ABB RobotStudio station: Workshop_RI.rspag

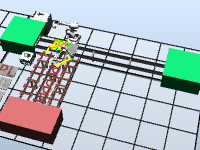
--- station ---
Station Workshop_RI (saved by RobotStudio format 3)
Controller IRB_1600_6kg_1.2m, task T_ROB1: task frame (RAPID world) sits at (2400, 1050, 0) mm, rotated rx 0 ry 0 rz -90 deg in the station
Controller IRB_140_6kg_0.81m, task T_ROB1: task frame (RAPID world) sits at (2400, -400, 420) mm in the station
Controller IRB_140_6kg_0.81m
  mechanical unit ROB_1: IRB140_6_81_C_03, 6 joints, base frame (0, 0, 0) mm
Controller IRB_1600_6kg_1.2m
  mechanical unit ROB_1: IRB1600_6_120__02, 6 joints, base frame (0, 0, 0) mm
Layout (positions relative to the parent item):
  - SC_SimpleVacuumGripper [protected smart component, left out]
  - Backup_Base_Parts [graphiccomponentgroup] at (1500, 500, 0) mm, rotated rx 0 ry 0 rz -90 deg
    - I_color [part] at (1567.69, 3594.7, 0) mm, rotated rx 0 ry 0 rz 90 deg
    - P_color [part] at (1567.69, 3594.7, 0) mm, rotated rx 0 ry 0 rz 90 deg
    - I_org [part] at (2207.69, 3594.7, 0) mm, rotated rx 0 ry 0 rz 90 deg
    - P_org [part] at (2207.69, 3594.7, 0) mm, rotated rx 0 ry 0 rz 90 deg
    - L_org [part] at (2207.69, 3594.7, 0) mm, rotated rx 0 ry 0 rz 90 deg
    - Base_org [part] at (2087.69, -1721.31, 0) mm
    - Base_holes [part] at (1447.69, -1721.31, 0) mm
    - L_color [part] at (1567.69, 3594.7, 0) mm, rotated rx 0 ry 0 rz 90 deg
  - SC_Main_Conveyor [protected smart component, left out]
  - Middle_PlaneSensor [smart component, from Libraries\PlaneSensor.rslib]
      properties: Origin=[2.865 -0.086804 0.458]; Axis1=[0 0.64 0]; Axis2=[0 0 0.05]; SensedPart=Base_holes_42
    - _sensorPart_ [part]
  - TempParts [graphiccomponentgroup]
    - Base_holes_42 [part] at (2866.18, 496.99, 457) mm, rotated rx 0 ry 0 rz 180 deg
    - Base_holes_1 [part] at (180, -43.01, 457) mm
  - SC_Letter_Conveyor_I [protected smart component, left out]
  - AW_Gun_PSF_25 [mechanism, from Tools\AW_Gun_PSF_25.rslib] at (1846.39, 1050, 893.77) mm, rotated rx -180 ry 60 rz 0 deg
  - Teste_Group1 [graphiccomponentgroup]
    - I_color_3 [part] at (7151.02, 376.99, 457) mm
    - L_color [part] at (7151.02, 376.99, 457) mm
    - P_color [part] at (7151.02, 376.99, 457) mm
    - Base_org_332 [part] at (2865, -43.01, 457) mm, rotated rx 0 ry 0 rz 90 deg
  - Teste_Group2 [graphiccomponentgroup] at (1650, 0, 0) mm
    - I_color_3 [part] at (7151.02, 376.99, 457) mm
    - L_color [part] at (7151.02, 376.99, 457) mm
    - P_color [part] at (7151.02, 376.99, 457) mm
    - Base_org_332 [part] at (2865, -43.01, 457) mm, rotated rx 0 ry 0 rz 90 deg
  - Furniture [graphiccomponentgroup]
    - Box_2 [part]
    - Box_3 [part]
    - Table [part] at (1825, -4950, 0) mm, rotated rx 0 ry 0 rz 90 deg
    - FlexPendant [part, from Equipment\FlexPendant.rslib] at (848.68, 1513.9, 739.04) mm, rotated rx -28.56 ry 0 rz 180 deg
    - IRC5_Compact [part, from Equipment\IRC5_Compact__02.rslib] at (772.3, -736.92, 0) mm
    - IRC5_Control-Module [part, from Equipment\IRC5_Control-Module.rslib] at (873.2, 1576.94, 100) mm, rotated rx 90 ry 0 rz 180 deg
    - FlexPendant_2 [part, from Equipment\FlexPendant.rslib] at (1028.44, -563.39, 415.73) mm, rotated rx -28.56 ry 0 rz 0 deg
  - IRB140_6_81_C_03 [mechanism, from Robots\IRB140_6_81_C_G_03.rslib] at (2400, -400, 420) mm; joint values [0, 0.4698, 0.3639, 0, 0.5236, 0] (rad or m)
  - SC_Letter_Conveyor_P [protected smart component, left out]
  - SC_Letter_Conveyor_L [protected smart component, left out]
  - Part_12 [part]
  - IRB1600_6_120__02 [mechanism, from Robots\IRB1600_6_120_G_02.rslib] at (2400, 1050, 0) mm, rotated rx 0 ry 0 rz -90 deg; joint values [-1.5708, -0.5581, 0.4967, 0, 0.5851, 0] (rad or m)
Attachment: SC_SimpleVacuumGripper is attached to IRB140_6_81_C_03 / Link6
Attachment: AW_Gun_PSF_25 is attached to IRB1600_6_120__02 / Link6
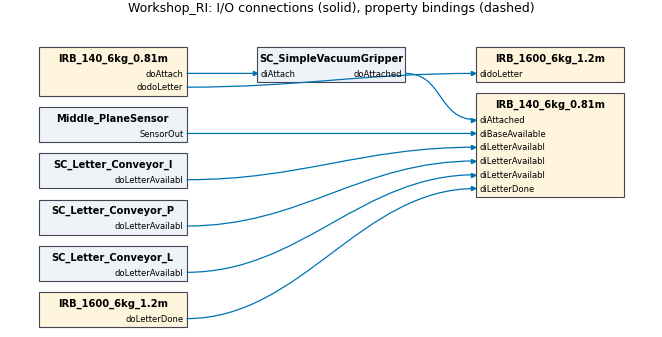
Station logic (signal -> signal, property => property):
  IRB_140_6kg_0.81m.doAttach -> SC_SimpleVacuumGripper.diAttach
  SC_SimpleVacuumGripper.doAttached -> IRB_140_6kg_0.81m.diAttached
  Middle_PlaneSensor.SensorOut -> IRB_140_6kg_0.81m.diBaseAvailable
  SC_Letter_Conveyor_I.doLetterAvailable -> IRB_140_6kg_0.81m.diLetterAvailable_I
  SC_Letter_Conveyor_P.doLetterAvailable -> IRB_140_6kg_0.81m.diLetterAvailable_P
  SC_Letter_Conveyor_L.doLetterAvailable -> IRB_140_6kg_0.81m.diLetterAvailable_L
  IRB_140_6kg_0.81m.dodoLetter -> IRB_1600_6kg_1.2m.didoLetter
  IRB_1600_6kg_1.2m.doLetterDone -> IRB_140_6kg_0.81m.diLetterDone

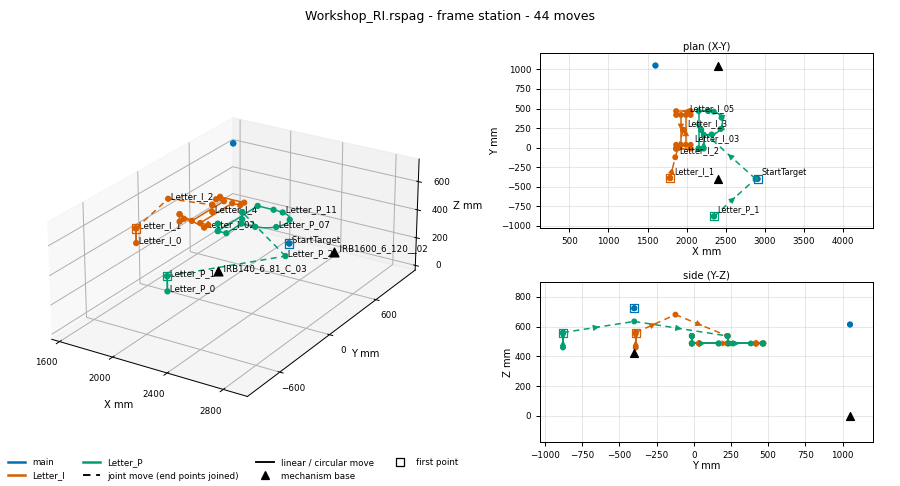
[picture p0: tool path of Workshop_RI.rspag in frame station, 44 of 44 moves have a stored position in this frame; points joined in program order, loops and branches not executed]
--- Backups/IRB_140_6kg_0.81m/RAPID/TASK1/PROGMOD/CalibData.mod ---
MODULE CalibData
	PERS tooldata SimpleVacuumGripper:=[TRUE,[[0,0,25],[1,0,0,0]],[0.5,[0,0,1],[1,0,0,0],0,0,0]];
ENDMODULE

--- Backups/IRB_140_6kg_0.81m/RAPID/TASK1/PROGMOD/Module1.mod ---
MODULE Module1
	CONST robtarget Letter_I_1:=[[-611.4,9.874,140],[0,-0.707106781,0.707106781,0],[1,0,0,0],[9E9,9E9,9E9,9E9,9E9,9E9]];
	CONST robtarget Letter_I_0:=[[-611.4,9.874,40],[0,-0.707106781,0.707106781,0],[1,0,0,0],[9E9,9E9,9E9,9E9,9E9,9E9]];
	CONST robtarget Letter_I_2:=[[-545.231385656,276.821478528,260.515371052],[-0.000000405,-0.529975894,0.848012707,-0.000000052],[1,0,0,0],[9E9,9E9,9E9,9E9,9E9,9E9]];
	CONST robtarget Letter_I_3:=[[-441.034,626.99,117],[0,1,0,0],[1,0,-1,0],[9E9,9E9,9E9,9E9,9E9,9E9]];
	CONST robtarget Letter_I_4:=[[-441.034,626.99,67],[0,1,0,0],[1,0,-1,0],[9E9,9E9,9E9,9E9,9E9,9E9]];
	CONST robtarget Letter_P_1:=[[-50,-479.055,140],[0,-0.707106781,0.707106781,0],[-2,0,1,0],[9E9,9E9,9E9,9E9,9E9,9E9]];
	CONST robtarget Letter_P_0:=[[-50,-479.055,40],[0,-0.707106781,0.707106781,0],[-2,0,1,0],[9E9,9E9,9E9,9E9,9E9,9E9]];
	CONST robtarget Letter_P_2:=[[481.657122129,0,215.039783495],[0.00000001,0.998648416,0.051974428,0.000000187],[0,-1,1,0],[9E9,9E9,9E9,9E9,9E9,9E9]];
	CONST robtarget Letter_P_3:=[[-213.633,626.99,117],[0,1,0,0],[1,0,3,0],[9E9,9E9,9E9,9E9,9E9,9E9]];
	CONST robtarget Letter_P_4:=[[-213.633,626.99,67],[0,1,0,0],[1,0,3,0],[9E9,9E9,9E9,9E9,9E9,9E9]];
    CONST robtarget StartPose:=[[507.45080207,0,303.659048752],[0.106520171,0,0.994310542,0],[0,0,0,0],[9E9,9E9,9E9,9E9,9E9,9E9]];
	CONST robtarget StartTarget:=[[507.45080207,0,303.659048752],[0.106520171,0,0.994310542,0],[0,0,0,0],[9E9,9E9,9E9,9E9,9E9,9E9]];
	PROC main()
        MoveJ StartTarget,v1000,z100,SimpleVacuumGripper\WObj:=wobj0;
        SetDO dodoLetter,0;
        WaitDI diLetterDone,0;
        Letter_I;
		Letter_P;
		Letter_L;
		MoveJ StartTarget,v1000,z100,SimpleVacuumGripper\WObj:=wobj0;
        SetDO dodoLetter,1;
        WaitDI diLetterDone,1;
    ENDPROC
    PROC Letter_I()
	    MoveJ Letter_I_1,v1000,z5,SimpleVacuumGripper\WObj:=wobj0;
	    MoveL Letter_I_0,v100,fine,SimpleVacuumGripper\WObj:=wobj0;
	    SetDO doAttach,1;
	    WaitDI diAttached,1;
	    MoveL Letter_I_1,v100,z10,SimpleVacuumGripper\WObj:=wobj0;
	    MoveJ Letter_I_2,v1000,z100,SimpleVacuumGripper\WObj:=wobj0;
	    MoveJ Letter_I_3,v1000,z5,SimpleVacuumGripper\WObj:=wobj0;
	    MoveL Letter_I_4,v100,fine,SimpleVacuumGripper\WObj:=wobj0;
	    SetDO doAttach,0;
	    WaitDI diAttached,0;
		MoveL Letter_I_3,v100,z5,SimpleVacuumGripper\WObj:=wobj0;
	ENDPROC
	PROC Letter_P()
	    MoveJ Letter_P_1,v1000,z5,SimpleVacuumGripper\WObj:=wobj0;
	    MoveL Letter_P_0,v100,fine,SimpleVacuumGripper\WObj:=wobj0;
	    SetDO doAttach,1;
	    WaitDI diAttached,1;
	    MoveL Letter_P_1,v100,z10,SimpleVacuumGripper\WObj:=wobj0;
	    MoveJ Letter_P_2,v1000,z10,SimpleVacuumGripper\WObj:=wobj0;
	    MoveJ Letter_P_3,v1000,z5,SimpleVacuumGripper\WObj:=wobj0;
	    MoveL Letter_P_4,v100,fine,SimpleVacuumGripper\WObj:=wobj0;
	    SetDO doAttach,0;
	    WaitDI diAttached,0;
		MoveL Letter_P_3,v100,z10,SimpleVacuumGripper\WObj:=wobj0;
	ENDPROC
	PROC Letter_L()
	ENDPROC
ENDMODULE

--- Backups/IRB_140_6kg_0.81m/RAPID/TASK1/SYSMOD/LINKEDM.sys ---
%%%
  VERSION:1
  LANGUAGE:ENGLISH
%%%

MODULE LINKEDM (SYSMODULE)

! FOLLOWER
!     Name of electronically linked follower axis used by operator at teach pendent.
      PERS string l_f_axis_name{5}       :=  ["",  "", "", "", ""];

!     Name of the mechanical unit for follower axis.
      PERS string l_f_mecunt_n{5}  :=  ["", "", "", "", ""];

!     Linked follower axis number in the mechanical unit (first axis in mech. unit is number 1).
      PERS num l_f_axis_no{5}      :=  [0,          0,   0,  0,  0];

! MASTER
!     Name of the mechanical unit for linked master axis.
      PERS string l_m_mecunt_n{5} :=  ["", "", "", "", ""];

!     Linked master axis number in the mechanical unit (first axis in mech. unit is number 1).
!     See axis number table in documentation for different master mechanical units.
      PERS num l_m_axis_no{5}     :=  [0,  0,  0,  0,  0];

! POSITION OFFSET
!     The increase of the allowed offset position between the master and follower
!     positions, used when starting AUTO mode. As soon as the offset is decreased
!     the old configurated parameter is used.
!     Example: 3 => the configurated value of allowed offset is increased 3 times.
      PERS num offset_ratio{5}       :=  [10,  10,   10,  10,  10];

! SPEED RATIO
!     Speed_ratio used in AUTO and JOG modes [ very_slow   slow    normal    fast]
!     Value 1 = max allowed manual speed.
      CONST num speed_ratio {20}      := [0.01, 0.01, 0.01, 0.01, 0.01,
                                          0.05, 0.05, 0.05, 0.05, 0.05,
                                          0.20, 0.20, 0.20, 0.20, 0.20,
                                          1.00, 1.00, 1.00, 1.00, 1.00];

! STEP SIZE
!     Displacement position used in JOG mode for each activation of positive or
!     negative movement.                  [very_short    short   normal   long]
!     Unit degees or meter.
      CONST num displacement {20}     := [0.001, 0.001, 0.001, 0.001, 0.001,
                                          0.005, 0.005, 0.005, 0.005, 0.005,
                                          0.020, 0.020, 0.020, 0.020, 0.020,
                                          0.100, 0.100, 0.100, 0.100, 0.100];


!-------------------------------------------------------------
 PROC Linked_m ()
      Linked_m_exe ;
 ENDPROC
ENDMODULE

--- Backups/IRB_1600_6kg_1.2m/RAPID/TASK1/PROGMOD/CalibData.mod ---
MODULE CalibData
	PERS tooldata AW_Gun:=[TRUE,[[119.5,0,352],[0.890213743,0,0.455543074,0]],[1,[0,0,100],[1,0,0,0],0,0,0]];
ENDMODULE

--- Backups/IRB_1600_6kg_1.2m/RAPID/TASK1/PROGMOD/Module1.mod ---
MODULE Module1
	CONST robtarget Letter_I_00:=[[1063.009551758,-533.999941406,537],[0,0,1,0],[-1,0,-1,0],[9E9,9E9,9E9,9E9,9E9,9E9]];
	CONST robtarget Letter_I_02:=[[1063.009551758,-348.068012719,487],[0,0,1,0],[-1,0,-1,0],[9E9,9E9,9E9,9E9,9E9,9E9]];
	CONST robtarget Letter_I_03:=[[1013.998206539,-348.068012719,487],[0,0,1,0],[-1,0,-1,0],[9E9,9E9,9E9,9E9,9E9,9E9]];
	CONST robtarget Letter_I_04:=[[1013.998206539,-409.137704777,487],[0,0,1,0],[-1,0,-1,0],[9E9,9E9,9E9,9E9,9E9,9E9]];
	CONST robtarget Letter_I_05:=[[632.020896977,-409.137704777,487],[0,0,1,0],[-1,0,-1,0],[9E9,9E9,9E9,9E9,9E9,9E9]];
	CONST robtarget Letter_I_06:=[[632.020896977,-348.068012719,487],[0,0,1,0],[-1,0,-1,0],[9E9,9E9,9E9,9E9,9E9,9E9]];
	CONST robtarget Letter_I_07:=[[583.009551758,-348.068012719,487],[0,0,1,0],[-1,0,-1,0],[9E9,9E9,9E9,9E9,9E9,9E9]];
	CONST robtarget Letter_I_08:=[[583.009551758,-533.999941406,487],[0,0,1,0],[-1,0,-1,0],[9E9,9E9,9E9,9E9,9E9,9E9]];
	CONST robtarget Letter_I_09:=[[632.020896977,-533.999941406,487],[0,0,1,0],[-1,0,-1,0],[9E9,9E9,9E9,9E9,9E9,9E9]];
	CONST robtarget Letter_I_10:=[[632.020896977,-472.930249348,487],[0,0,1,0],[-1,0,-1,0],[9E9,9E9,9E9,9E9,9E9,9E9]];
	CONST robtarget Letter_I_11:=[[1013.998206539,-472.930249348,487],[0,0,1,0],[-1,0,-1,0],[9E9,9E9,9E9,9E9,9E9,9E9]];
	CONST robtarget Letter_I_12:=[[1013.998206539,-533.999941406,487],[0,0,1,0],[-1,0,-1,0],[9E9,9E9,9E9,9E9,9E9,9E9]];
	CONST robtarget Letter_I_01:=[[1063.009551758,-533.999941406,487],[0,0,1,0],[-1,0,-1,0],[9E9,9E9,9E9,9E9,9E9,9E9]];
	CONST robtarget Letter_P_00:=[[1063.009551758,-245.528012719,537],[0,0,1,0],[-1,0,-1,0],[9E9,9E9,9E9,9E9,9E9,9E9]];
	CONST robtarget Letter_P_01:=[[1063.009551758,-245.528012719,487],[0,0,1,0],[-1,0,-1,0],[9E9,9E9,9E9,9E9,9E9,9E9]];
	CONST robtarget Letter_P_02:=[[1063.009551758,-181.735468149,487],[0,0,1,0],[-1,0,-1,0],[9E9,9E9,9E9,9E9,9E9,9E9]];
	CONST robtarget Letter_P_03:=[[884.079243816,-181.735468149,487],[0,0,1,0],[-1,0,-1,0],[9E9,9E9,9E9,9E9,9E9,9E9]];
	CONST robtarget Letter_P_04:=[[884.079243816,-127.667396836,487],[0,0,1,0],[-1,0,-1,0],[9E9,9E9,9E9,9E9,9E9,9E9]];
	CONST robtarget Letter_P_05:=[[880.918790007,-80.746813367,487],[0,0,1,0],[-1,0,-1,0],[9E9,9E9,9E9,9E9,9E9,9E9]];
	CONST robtarget Letter_P_06:=[[855.829649003,-11.216829575,487],[0,0,1,0],[-1,0,-1,0],[9E9,9E9,9E9,9E9,9E9,9E9]];
	CONST robtarget Letter_P_07:=[[812.701610105,33.515747411,487],[0,0,1,0],[0,-1,0,0],[9E9,9E9,9E9,9E9,9E9,9E9]];
	CONST robtarget Letter_P_08:=[[743.07438158,57.182684202,487],[0,0,1,0],[0,-1,0,0],[9E9,9E9,9E9,9E9,9E9,9E9]];
	CONST robtarget Letter_P_09:=[[666.679527447,46.260885174,487],[0,0,1,0],[0,-1,0,0],[9E9,9E9,9E9,9E9,9E9,9E9]];
	CONST robtarget Letter_P_10:=[[612.960929392,0.695650166,487],[0,0,1,0],[0,-1,0,0],[9E9,9E9,9E9,9E9,9E9,9E9]];
	CONST robtarget Letter_P_11:=[[590.011172503,-52.205484356,487],[0,0,1,0],[-1,0,-1,0],[9E9,9E9,9E9,9E9,9E9,9E9]];
	CONST robtarget Letter_P_12:=[[584.759956944,-85.365938165,487],[0,0,1,0],[-1,0,-1,0],[9E9,9E9,9E9,9E9,9E9,9E9]];
	CONST robtarget Letter_P_13:=[[583.009551758,-124.944544324,487],[0,0,1,0],[-1,0,-1,0],[9E9,9E9,9E9,9E9,9E9,9E9]];
	CONST robtarget Letter_P_14:=[[583.009551758,-245.528012719,487],[0,0,1,0],[-1,0,-1,0],[9E9,9E9,9E9,9E9,9E9,9E9]];
	CONST robtarget StartTarget:=[[0.000250725,-798.69947369,614.279917089],[0.035775265,0.706201086,0.706201308,-0.035775276],[-1,-1,-1,0],[9E9,9E9,9E9,9E9,9E9,9E9]];
	PROC main()
        MoveJ StartTarget,v1000,z100,AW_Gun\WObj:=wobj0;
        SetDO doLetterDone,0;
        WaitDI didoLetter,0;
        WaitDI didoLetter,1;
        Letter_I;
        Letter_P;
        Letter_L;
        MoveJ StartTarget,v1000,z100,AW_Gun\WObj:=wobj0;
        SetDO doLetterDone,0;

    ENDPROC
    PROC Letter_I()
	    MoveJ Letter_I_00,v1000,z5,AW_Gun\WObj:=wobj0;
	    MoveL Letter_I_02,v200,z0,AW_Gun\WObj:=wobj0;
	    MoveL Letter_I_03,v200,z0,AW_Gun\WObj:=wobj0;
	    MoveL Letter_I_04,v200,z0,AW_Gun\WObj:=wobj0;
	    MoveL Letter_I_05,v200,z0,AW_Gun\WObj:=wobj0;
	    MoveL Letter_I_06,v200,z0,AW_Gun\WObj:=wobj0;
	    MoveL Letter_I_07,v200,z0,AW_Gun\WObj:=wobj0;
	    MoveL Letter_I_08,v200,z0,AW_Gun\WObj:=wobj0;
	    MoveL Letter_I_09,v200,z0,AW_Gun\WObj:=wobj0;
	    MoveL Letter_I_10,v200,z0,AW_Gun\WObj:=wobj0;
	    MoveL Letter_I_11,v200,z0,AW_Gun\WObj:=wobj0;
	    MoveL Letter_I_12,v200,z0,AW_Gun\WObj:=wobj0;
	    MoveL Letter_I_01,v200,z0,AW_Gun\WObj:=wobj0;
	    MoveL Letter_I_00,v200,z10,AW_Gun\WObj:=wobj0;
	ENDPROC
	PROC Letter_P()
	    MoveJ Letter_P_00,v1000,z5,AW_Gun\WObj:=wobj0;
	    MoveL Letter_P_01,v100,z0,AW_Gun\WObj:=wobj0;
	    MoveL Letter_P_02,v100,z0,AW_Gun\WObj:=wobj0;
	    MoveL Letter_P_03,v100,z0,AW_Gun\WObj:=wobj0;
	    MoveC Letter_P_04,Letter_P_05,v100,z0,AW_Gun\WObj:=wobj0;
	    MoveC Letter_P_06,Letter_P_07,v100,z0,AW_Gun\WObj:=wobj0;
	    MoveC Letter_P_08,Letter_P_09,v100,z0,AW_Gun\WObj:=wobj0;
	    MoveC Letter_P_10,Letter_P_11,v100,z0,AW_Gun\WObj:=wobj0;
	    MoveC Letter_P_12,Letter_P_13,v100,z0,AW_Gun\WObj:=wobj0;
	    MoveL Letter_P_14,v100,z0,AW_Gun\WObj:=wobj0;
	    MoveL Letter_P_01,v100,z0,AW_Gun\WObj:=wobj0;
	    MoveL Letter_P_00,v200,z10,AW_Gun\WObj:=wobj0;
	ENDPROC
	PROC Letter_L()
	ENDPROC
ENDMODULE

--- Backups/IRB_140_6kg_0.81m/SYSPAR/EIO.cfg ---
EIO:CFG_1.0:6:1::
#
EIO_SIGNAL:

      -Name "diAttached" -SignalType "DI" -Access "All"

      -Name "diBaseAvailable" -SignalType "DI" -Access "All"

      -Name "diLetterAvailable_I" -SignalType "DI" -Access "All"

      -Name "doAttach" -SignalType "DO" -Access "All"

      -Name "doMove" -SignalType "DO" -Access "All"

      -Name "diLetterAvailable_P" -SignalType "DI" -Access "All"

      -Name "diLetterAvailable_L" -SignalType "DI" -Access "All"

      -Name "dodoLetter" -SignalType "DO" -Access "All"

      -Name "diLetterDone" -SignalType "DI" -Access "All"

--- Backups/IRB_1600_6kg_1.2m/SYSPAR/EIO.cfg ---
EIO:CFG_1.0:6:1::
#
EIO_SIGNAL:

      -Name "didoLetter" -SignalType "DI" -Access "All"

      -Name "doLetterDone" -SignalType "DO" -Access "All"
